TYPE sEL1809 :
STRUCT
	ch1  :BOOL;
	ch2  :BOOL;
	ch3  :BOOL;
	ch4  :BOOL;
	ch5  :BOOL;
	ch6  :BOOL;
	ch7  :BOOL;
	ch8  :BOOL;
	ch9  :BOOL;
	ch10  :BOOL;
	ch11  :BOOL;
	ch12  :BOOL;
	ch13  :BOOL;
	ch14  :BOOL;
	ch15  :BOOL;
	ch16  :BOOL;
END_STRUCT
END_TYPE

(* stored: Version 1.1.0.1, ProductVersion 3.1.4024.12
   DUT sEL1809: Id {a3d8ce42-f463-454f-b6ff-78e3e3c8d850} *)
